{attribute 'GeneratedUsingTerminal: EK1122-0000-0018'}
{attribute addProperty BoxType "EK1122-0000-0018"}
{attribute addProperty Id "Beckhoff_EL6xxxsub_EK1100EK1100_1FC0878B2"}
{attribute addProperty CRC "3058719422"}
{attribute addProperty Size "2"}
TYPE Beckhoff_EL6xxxEK1122_B6505ABE EXTENDS EK1122_1FC0878B :
STRUCT
	{attribute addProperty Name "Beckhoff EL6xxxsub EK1100"}
	{attribute addProperty PreviousPort "Beckhoff EL6xxxEK1122 : D"}
	Beckhoff_EL6xxxsub_EK1100 : EK1100_1FC0878B;
END_STRUCT
END_TYPE

(* stored: Version 1.2.0.0, ProductVersion 3.1.4024.9
   DUT Beckhoff_EL6xxxEK1122_B6505ABE: Id {5311389d-5ddf-4d9c-b2e1-795a16968bb1} *)
